PROGRAM BackgroundRS232
VAR
	
END_VAR

GVL_IO.stSerialData_S02_S04.fbSerialCom(RxBufferEL:=GVL_IO.stSerialData_S02_S04.RxBufferEL,TxBufferEL:=GVL_IO.stSerialData_S02_S04.TxBufferEL);
MAIN.fbWeighingTunel.fbWeighingStation.fbWeighing();

END_PROGRAM

(* stored: Version 1.1.0.1, ProductVersion 3.1.4024.16
   POU BackgroundRS232: Id {9a20473f-0d3f-4584-b429-33e10587a848}, SpecialFunc None *)
